{attribute 'GeneratedUsingTerminal: EL4038-0000-0016'}
{attribute addProperty BoxType "EL4038-0000-0016"}
{attribute addProperty Description "EL4038 8Ch. Ana. Output +/-10V, 12bit"}
{attribute addProperty Physics "KK"}
{attribute addProperty Id "AO_Outputs_Channel_1AT %Q*AO_Output_Channel_BA7EBB7C2AO_Outputs_Channel_2AT %Q*AO_Output_Channel_BA7EBB7C2AO_Outputs_Channel_3AT %Q*AO_Output_Channel_BA7EBB7C2AO_Outputs_Channel_4AT %Q*AO_Output_Channel_BA7EBB7C2AO_Outputs_Channel_5AT %Q*AO_Output_Channel_BA7EBB7C2AO_Outputs_Channel_6AT %Q*AO_Output_Channel_BA7EBB7C2AO_Outputs_Channel_7AT %Q*AO_Output_Channel_BA7EBB7C2AO_Outputs_Channel_8AT %Q*AO_Output_Channel_BA7EBB7C2WcStateAT %I*WcState_0B2B16F91InfoDataAT %I*InfoData_32EB74EA10"}
{attribute addProperty CRC "1316477058"}
{attribute addProperty Size "27"}
TYPE EL4038_4E77D882 EXTENDS EtcSlaveTerminalBase_947E5A46 :
STRUCT
	{attribute addProperty Name "AO_Outputs_Channel_1"}
	AO_Outputs_Channel_1 : AO_Output_Channel_BA7EBB7C;
	{attribute addProperty Name "AO_Outputs_Channel_2"}
	AO_Outputs_Channel_2 : AO_Output_Channel_BA7EBB7C;
	{attribute addProperty Name "AO_Outputs_Channel_3"}
	AO_Outputs_Channel_3 : AO_Output_Channel_BA7EBB7C;
	{attribute addProperty Name "AO_Outputs_Channel_4"}
	AO_Outputs_Channel_4 : AO_Output_Channel_BA7EBB7C;
	{attribute addProperty Name "AO_Outputs_Channel_5"}
	AO_Outputs_Channel_5 : AO_Output_Channel_BA7EBB7C;
	{attribute addProperty Name "AO_Outputs_Channel_6"}
	AO_Outputs_Channel_6 : AO_Output_Channel_BA7EBB7C;
	{attribute addProperty Name "AO_Outputs_Channel_7"}
	AO_Outputs_Channel_7 : AO_Output_Channel_BA7EBB7C;
	{attribute addProperty Name "AO_Outputs_Channel_8"}
	AO_Outputs_Channel_8 : AO_Output_Channel_BA7EBB7C;
	{attribute addProperty Name "WcState"}
	WcState : WcState_0B2B16F9;
	{attribute addProperty Name "InfoData"}
	InfoData : InfoData_32EB74EA;
END_STRUCT
END_TYPE

(* stored: Version 1.2.0.0, ProductVersion 3.1.4024.11
   DUT EL4038_4E77D882: Id {73ae9652-cd78-4bc0-9972-dc111ca5a485} *)
